PROGRAM MAIN
VAR	
	unixTime: UnixTimestamp;
	timestampNanoseconds: ULINT;

	// General variables
	mxReset									: BOOL;
	mxEmergency								: BOOL;
	EmButtons								: BOOL;
	mxAutoMode								: BOOL; (* "1" = Auto, "0" = Manual *)
	mxFirstCycle							: BOOL;
	mxErrorInit								: BOOL;
	mxInitialized							: BOOL;
	SR_AttemptedStartWithNoProductLoaded	: SR;
	
	// Sub objects
	InMoldDrying							: FB_InMoldDrying;
	ProductHandling							: FB_ProductHandling;
	Blink									: FB_Blink;

	// Variables for parameter structs and error structs
	ComSC									: ST_Com_SpeedControl;	// Communication struct for speedcontrol
	MachPar									: ST_MachPar;
	ProductPar								: ST_ProdPar;
	SysPar									: ST_SysPar;
	Errors									: ST_Errors;
	OEEpar									: ST_OEE;
	
	// Variables for/with HMI purposes
{Region "HMI variables"}
	mxHMI_Start								: BOOL;
	mxHMI_Stop								: BOOL;
	mxHMI_Pause								: BOOL;
	mxHMI_Sample							: BOOL;
	mxHMI_Reset								: BOOL;
	mxHMI_StartInit							: BOOL;
	mxHMI_StopInit							: BOOL;
	mxHMI_EnableHeating						: BOOL;

	mxHMI_StartState						: BOOL;
	mxHMI_StopState							: BOOL;
	mxHMI_PauseState						: BOOL;
	mxHMI_SampleState						: BOOL;
	mxHMI_Stopping							: BOOL;
	mxHMI_StartHydraulicsState				: BOOL;
	mxHMI_StopHydraulicsState				: BOOL;
	mxHMI_StartHydraulics					: BOOL;
	mxHMI_StopHydraulics					: BOOL;
	mxHydraulicsReady						: BOOL;
	mxProductLoaded							: BOOL;
	mxMachineInRest							: BOOL;
	
	// Speedcontrol states for hmi
	mrHMI_SpeedControlModulo				: LREAL;
	mxHMI_StartFormingPulse					: BOOL;
	mxHMI_StopFormingPulse					: BOOL;
	mxHMI_SlotANotFree						: BOOL;
	mxHMI_SlotBNotFree						: BOOL;
	mxHMI_IMDHasES							: BOOL;
	mrHMI_MaximumNrOfKickoffs				: REAL;
	mrHMI_ActNrOfKickoffs					: REAL;
	mxHMI_IMDRTO							: BOOL;
	mxHMI_IMDStopped						: BOOL;
	mxHMI_IMDRunning						: BOOL;
	mrHMI_DictatedKoSpeedControl			: LREAL;
	
	
	T_HMIReset								: TON;
	FT_AutoMode								: F_Trig;
	RT_MasterReset							: R_trig;
{End region}
	
	// Triggers for starting and stopping
	RT_Start								: R_TRIG;
	RT_Stop									: R_TRIG;
	RT_StopBySC								: R_TRIG;
	RT_StartBySC							: R_TRIG;
	RT_Pause								: R_TRIG;
	RT_StartInit							: R_TRIG;
	RT_StopInit								: R_TRIG;
	RT_StopOnLowLvl							: R_TRIG;
	RT_StartHydraulics						: R_TRIG;
	RT_StopHydraulics						: R_TRIG;	

	RT_PauseReqGantryA						: R_TRIG;
	RT_PauseReqGantryB						: R_TRIG;
	RT_PauseReqProdHandling					: R_TRIG;
	RT_PauseReqImd							: R_TRIG;
	
	// 24Volt error
	ix24VoltError1							AT %I* : BOOL;
	ix24VoltError2							AT %I* : BOOL;
	SR_24VError1							: SR;
	SR_24VError2							: SR;	
	
	// inputs and ouputs regarding safety 
{Region "Safety variables"}
	ixTwinSafe_SafetyRelay 					AT %I*:ARRAY[1..GVL.MAX_ZONES] OF BOOL; (* couple to zones in Safety programm FB outputs *)
	qxTwinSafe_Reset						AT %Q*: BOOL;
	FbError 								AT %I*: BOOL;
	ComErr 									AT %I*: BOOL;
	OutErr 									AT %I*: BOOL;
	
	(* Operator side/Front *)
	ixResetImdFront							AT %I* : BOOL;
	ixDoorReqImdFront						AT %I* : BOOL;
	qxLightEmStopImdFront					AT %Q* : BOOL;
	qxLightDoorReqImdFront					AT %Q* : BOOL;
	ixEmStopImdFront						AT %I* 	: ARRAY[0..1] OF BOOL; (* couple to the TwinSAFE inputs *)
	(* NON Operator side/Back *)
	ixResetImdBack							AT %I* : BOOL;
	ixDoorReqImdBack						AT %I* : BOOL;
	qxLightEmStopImdBack					AT %Q* : BOOL;
	qxLightDoorReqImdBack					AT %Q* : BOOL;
	ixEmStopImdBack							AT %I* 	: ARRAY[0..1] OF BOOL; (* couple to the TwinSAFE inputs *)

	(* Safety door switches *)
	ixSafetyFrontDoorLeft					AT %I* 	: ARRAY[0..1] OF BOOL; (* couple to the TwinSAFE inputs *)
	ixSafetyFrontDoorMiddle					AT %I* 	: ARRAY[0..1] OF BOOL; (* couple to the TwinSAFE inputs *)
	ixSafetyFrontDoorRight					AT %I* 	: ARRAY[0..1] OF BOOL; (* couple to the TwinSAFE inputs *)
	ixSafetyBackDoorLeft1					AT %I* 	: ARRAY[0..1] OF BOOL; (* couple to the TwinSAFE inputs *)
	ixSafetyBackDoorLeft2					AT %I* 	: ARRAY[0..1] OF BOOL; (* couple to the TwinSAFE inputs *)
	ixSafetyBackDoorMiddle3					AT %I* 	: ARRAY[0..1] OF BOOL; (* couple to the TwinSAFE inputs *)
	ixSafetyBackDoorMiddle4					AT %I* 	: ARRAY[0..1] OF BOOL; (* couple to the TwinSAFE inputs *)
	ixSafetyBackDoorRight5					AT %I* 	: ARRAY[0..1] OF BOOL; (* couple to the TwinSAFE inputs *)
	ixSafetyBackDoorRight6					AT %I* 	: ARRAY[0..1] OF BOOL; (* couple to the TwinSAFE inputs *)

	ixResetGantryA_Front					AT %I* : BOOL;
	ixDoorReqGantryA_Front					AT %I* : BOOL;
	qxLightEmStopGantryA_Front				AT %Q* : BOOL;
	qxLightDoorReqGantryA_Front				AT %Q* : BOOL;
	ixEmStopGantryA_Front					AT %I* 	: ARRAY[0..1] OF BOOL; (* couple to the TwinSAFE inputs *)

	ixResetGantryA_Back						AT %I* : BOOL;
	ixDoorReqGantryA_Back					AT %I* : BOOL;
	qxLightEmStopGantryA_Back				AT %Q* : BOOL;
	qxLightDoorReqGantryA_Back				AT %Q* : BOOL;
	ixEmStopGantryA_Back					AT %I* 	: ARRAY[0..1] OF BOOL; (* couple to the TwinSAFE inputs *)

	ixResetGantryB_Front					AT %I* : BOOL;
	ixDoorReqGantryB_Front					AT %I* : BOOL;
	qxLightEmStopGantryB_Front				AT %Q* : BOOL;
	qxLightDoorReqGantryB_Front				AT %Q* : BOOL;
	ixEmStopGantryB_Front					AT %I* 	: ARRAY[0..1] OF BOOL; (* couple to the TwinSAFE inputs *)

	ixResetGantryB_Back						AT %I* : BOOL;
	ixDoorReqGantryB_Back					AT %I* : BOOL;
	qxLightEmStopGantryB_Back				AT %Q* : BOOL;
	qxLightDoorReqGantryB_Back				AT %Q* : BOOL;
	ixEmStopGantryB_Back					AT %I* 	: ARRAY[0..1] OF BOOL; (* couple to the TwinSAFE inputs *)
	
	ixSafetyGantryA_FrontDoorLeft			AT %I* 	: ARRAY[0..1] OF BOOL; (* couple to the TwinSAFE inputs *)
	ixSafetyGantryA_FrontDoorRight			AT %I* 	: ARRAY[0..1] OF BOOL; (* couple to the TwinSAFE inputs *)
	ixSafetyGantryA_BackDoor				AT %I* 	: ARRAY[0..1] OF BOOL; (* couple to the TwinSAFE inputs *)
	ixSafetyGantryB_FrontDoorLeft			AT %I* 	: ARRAY[0..1] OF BOOL; (* couple to the TwinSAFE inputs *)
	ixSafetyGantryB_FrontDoorRight			AT %I* 	: ARRAY[0..1] OF BOOL; (* couple to the TwinSAFE inputs *)
	ixSafetyGantryB_BackDoor				AT %I* 	: ARRAY[0..1] OF BOOL; (* couple to the TwinSAFE inputs *)
{End Region}
	
	// Emergency stops
	SR_exEmergency							: ARRAY[1..GVL.MAX_ZONES] OF SR; (* Emergency of the zones *)
	SR_EmStopImdFront						: SR;
	SR_EmStopImdBack						: SR;
	SR_EmStopGantryA_Front					: SR;
	SR_EmStopGantryA_Back					: SR;
	SR_EmStopGantryB_Front					: SR;
	SR_EmStopGantryB_Back					: SR;
	
	// Emergency Doors IMD
	SR_SafetyFrontDoorLeft					: SR;
	SR_SafetyFrontDoorMiddle				: SR;
	SR_SafetyFrontDoorRight					: SR;
	SR_SafetyBackDoorLeft1					: SR;
	SR_SafetyBackDoorLeft2					: SR;
	SR_SafetyBackDoorMiddle3				: SR;
	SR_SafetyBackDoorMiddle4				: SR;
	SR_SafetyBackDoorRight5					: SR;
	SR_SafetyBackDoorRight6					: SR;
	DoorRequestImdFront						: GateRequest;
	DoorRequestImdBack						: GateRequest;
	DoorRequestGantryAFront					: GateRequest;
	DoorRequestGantryABack					: GateRequest;
	DoorRequestGantryBFront					: GateRequest;
	DoorRequestGantryBBack					: GateRequest;
	
	// Emergency Doors Gantries
	SR_SafetyGantryA_FrontDoorLeft			: SR;	
	SR_SafetyGantryA_FrontDoorRight			: SR;
	SR_SafetyGantryA_BackDoor				: SR;
	SR_SafetyGantryB_FrontDoorLeft			: SR;	
	SR_SafetyGantryB_FrontDoorRight			: SR;
	SR_SafetyGantryB_BackDoor				: SR;

	// Presistent data
	ChkMachPar								: ST_MachPar;
	CmpMachPar								: DINT;
	ChkSysPar								: ST_SysPar;
	CmpSysPar								: DINT;
	RTRIG_WritePersistent					: R_TRIG;
	FB_WritePersistentData					:  WritePersistentData;
	FB_GetCurTaskIdx						: GETCURTASKINDEX;
	T_WritePersistent						: TON;
	
	// Variables for the ethercat diagnosing.
	iwDevID									AT %I* :UINT;
	iAmsNetID								AT %I* :ARRAY [0..5] OF BYTE;
	iwSlaveCount							AT %I* :UINT;
	iwCfgSlaveCount							AT %I* :UINT;
	iwDevState								AT %I* :UINT;
	EtherCatDiag							:FB_EtherCATDiag;
	AmsNetID								: STRING;
	DeviceID								: INT;
	
	PlcCycleTime     						: REAL := 10.0;
	
	// Variables for O.E.E
	L1										AT %I* : ST_PowerMeasurement;
	L2										AT %I* : ST_PowerMeasurement;
	L3										AT %I* : ST_PowerMeasurement;	
	ActNrOfKickoffs							: REAL;	
	oldSecond								: INT;
	NTGetTime								: NT_GetTime;
	mxPulseCycle							: BOOL; 				(* Pulse 1 cycle on, 1 cycle off *)
	SysTime									: TIMESTRUCT;
	RT_1SecondTrigger						: R_TRIG;
	
	// Outputs for alarm tower.
	qxLightGreen							AT %Q* : BOOL;
	qxLightYellow							AT %Q* : BOOL;
	qxLightRed								AT %Q* : BOOL;
	qxAlarmHorn								AT %Q* : BOOL;
	
	// Variables for the UPS
	ixMainSwitchOFF							AT %I* : BOOL;	
	ixUPS_Alarm								AT %I* : BOOL;
	ixUPS_BatMode							AT %I* : BOOL;
	ixUPS_Charge							AT %I* : BOOL;
	qxPcRemoteOff							AT %Q* : BOOL;
	T_BatteryMode							: TON;
	T_MaintSwitch							: TON;
	SR_UPSAlarm								: SR;
	mxEmDoors								: BOOL;


	mxIMDUnlocked							: BOOL;
	mxProdHandlingUnlocked					: BOOL;
	mxEmptyByStopSC							: BOOL;

	RT_Sample: R_TRIG;
	mxSample: BOOL;
	RT_RestartAfterDoorOpened: R_TRIG;
	FT_Sample: F_TRIG;
	
	mxReset_ByStartInmold			: BOOL;
	mxReset_ByStartProdHandling		: BOOL;
	RT_InMoldDryingBusy				: R_TRIG;
	RT_ProdHandlingBusy				: R_TRIG;
	
	//Main Air supply
	MainAirSupply					: FB_MonoValveNoFdbck;
	MainAirPressureSwitch	AT %I* 	: BOOL;
	SR_MainAirPressureError			: SR;
	
END_VAR

unixTime();
//timestampMilliseconds := unixTime.milliseconds;
//timestampSeconds := unixTime.seconds;
timestampNanoseconds := unixTime.nanoseconds;

// 					Object Calls				//
FB_GetCurTaskIdx();
mxFirstCycle:= _TaskInfo[FB_GetCurTaskIdx.index].FirstCycle;
PlcCycleTime:= UDINT_TO_REAL(_TaskInfo[FB_GetCurTaskIdx.index].CycleTime/10000);
RemanentData();
Blink();
Objects();
HMIState();

// 					R_Trigs.					//
RT_StartHydraulics(CLK:= mxHMI_StartHydraulics);
RT_StopHydraulics(CLK:= mxHMI_StopHydraulics);
RT_Start(CLK:= mxHMI_Start);// OR (ComSC.SpeedControl_IMD.StartForming AND NOT InMoldDrying.mxInPause));
RT_Stop(CLK:= mxHMI_Stop); 
RT_StartBySC(CLK:= ComSC.SpeedControl_IMD.StartFormingA OR ComSC.SpeedControl_IMD.StartFormingB);
RT_StopBySC(CLK:= ComSC.SpeedControl_IMD.StopForming); 
RT_StopOnLowLvl(CLK:= Main.Errors.InMoldDryingErrors.ProductForming.LowLvlOnBothTanks);
RT_Pause(CLK:= mxHMI_Pause);
RT_Sample(CLK:=mxHMI_Sample);
FT_Sample(CLK:=InMoldDrying.mxSample);
RT_StartInit(CLK:= mxHMI_StartInit);
RT_StopInit(CLK:= mxHMI_StopInit);
RT_MasterReset(CLK:= NOT mxAutoMode);
mxInitialized:= InMoldDrying.mxInitialized AND ProductHandling.mxInitialized;
mxMachineInRest := NOT InMoldDrying.mxCycleBusy AND NOT ProductHandling.mxCycleBusy;


// 					Start the Hydraulics		//
IF (RT_StartHydraulics.Q OR (RT_RestartAfterDoorOpened.Q AND InMoldDrying.HydraulicsMain.mxCycleInPause AND mxAutoMode)) AND NOT mxErrorInit THEN
	InMoldDrying.M_StartHydraulics();
END_IF

// 					Stop hydraulics
IF RT_StopHydraulics.Q THEN
	InMoldDrying.M_StopHydraulics();
END_IF

RT_InMoldDryingBusy(CLK:=InMoldDrying.mxCycleBusy);
RT_ProdHandlingBusy(CLK:=ProductHandling.mxCycleBusy);
IF RT_InMoldDryingBusy.Q THEN
	mxReset_ByStartInmold := TRUE;
END_IF
IF RT_ProdHandlingBusy.Q THEN
	mxReset_ByStartProdHandling := TRUE;
END_IF
IF NOT mxEmptyByStopSC THEN
	mxReset_ByStartInmold := FALSE;
	mxReset_ByStartProdHandling := FALSE;	
END_IF

// 					Start machine				//
IF (RT_Start.Q OR (mxEmptyByStopSC AND NOT ComSC.SpeedControl_IMD.StopForming)) AND mxAutoMode AND mxInitialized AND NOT mxErrorInit AND mxProductLoaded AND mxHydraulicsReady AND NOT mxIMDUnlocked AND NOT mxProdHandlingUnlocked THEN  
	InMoldDrying.M_StartCycle(); 
	ProductHandling.M_StartCycle();
	mxHMI_Stopping :=FALSE;
	IF mxReset_ByStartInmold AND mxReset_ByStartProdHandling THEN
		mxEmptyByStopSC := FALSE;
	END_IF
END_IF

//					IMD Pause (stopinpos)		//
IF RT_PauseReqImd.Q THEN
	InMoldDrying.M_StopCycle();	
	mxEmptyByStopSC := FALSE;
END_IF

//					Producthandling Pause (stopinpos)		//
IF RT_PauseReqProdHandling.Q THEN
	ProductHandling.M_StopCycle();	
	mxEmptyByStopSC := FALSE;
END_IF

//					Normal stop					//
IF ((RT_StopOnLowLvl.Q OR RT_Stop.Q OR RT_StopBySC.Q) AND mxAutoMode) THEN  
	InMoldDrying.M_StopCycleEmpty();  
	Producthandling.M_StopCycleEmpty(); 
	mxHMI_Stopping := TRUE;		
	mxEmptyByStopSC := FALSE;
	IF 	RT_StopBySC.Q AND (ProductHandling.mxCycleBusy OR InMoldDrying.mxCycleBusy) THEN
		mxEmptyByStopSC := TRUE;
	END_IF			
END_IF

//					Init machine				//
IF RT_StartInit.Q AND mxAutoMode AND mxProductLoaded AND NOT mxErrorInit AND mxHydraulicsReady THEN 
	InMoldDrying.M_StartInit(); 
	mxEmptyByStopSC := FALSE;
	Producthandling.M_StartInit(); 
END_IF
IF RT_StopInit.Q OR mxErrorInit THEN
	InMoldDrying.M_StopInit();
	ProductHandling.M_StopInit();
	mxEmptyByStopSC := FALSE;
END_IF

//					Stop direct error			//
IF mxErrorInit OR InMoldDrying.mxErrorInit OR ProductHandling.Errors.Gantry_A.Collision OR ProductHandling.Errors.Gantry_B.Collision THEN
	InMoldDrying.M_StopDirect();
	mxEmptyByStopSC := FALSE;
END_IF

IF mxErrorInit OR ProductHandling.mxErrorInit THEN
	ProductHandling.M_StopDirect();
	mxEmptyByStopSC := FALSE;
END_IF



//					Signal light				//
qxLightEmStopImdFront:= qxLightEmStopImdBack:= qxLightEmStopGantryA_Front:= qxLightEmStopGantryA_Back:= qxLightEmStopGantryB_Front:= qxLightEmStopGantryB_Back := 
	Errors.exEmergency[1] OR Errors.exEmergency[2] OR Errors.exEmergency[3] OR Errors.exEmergency[4] OR Errors.exEmergency[5] OR Errors.exEmergency[6] OR Errors.exEmergency[7];
qxLightRed:= HMI.mxError;
qxLightGreen:= mxHMI_StartState := (InMoldDrying.mxCycleBusy OR ProductHandling.mxCycleBusy) AND NOT mxHMI_PauseState;
qxLightYellow:= FALSE;

//					Reseting					//
T_HMIReset(IN:= mxHMI_Reset,PT:=T#1S);
IF T_hmiReset.Q THEN mxHMI_Reset:=FALSE; END_IF

mxReset:= qxTwinSafe_Reset:= mxHMI_Reset OR ixResetImdFront OR ixResetImdBack OR ixResetGantryA_Front OR ixResetGantryA_Back OR ixResetGantryB_Front OR ixResetGantryB_Back;

//					Master reset				//
IF RT_MasterReset.Q THEN
	InMoldDrying.mxResetCycleState := TRUE;
	InMoldDrying.mxResetInitState := TRUE;
	ProductHandling.mxResetCycleState:= TRUE;
	ProductHandling.mxResetInitState:= TRUE;
	mxEmptyByStopSC := FALSE;
END_IF

// 					Sample button				//
IF RT_Sample.Q THEN
	mxSample:= InMoldDrying.mxSample := TRUE;
END_IF; 

IF FT_Sample.Q THEN
	mxSample:=FALSE;
END_IF


// Get AMS net id and device id for ethercat topology
AmsNetID:= F_CreateAmsNetId(iAmsNetID);
DeviceID:= UINT_TO_INT(iwDevID);

// 					Force HMI bits to zero		//
mxHMI_Start := FALSE;
mxHMI_Stop := FALSE;
mxHMI_Pause := FALSE;
mxHMI_Sample:=FALSE;
mxHMI_StartHydraulics := FALSE;
mxHMI_StopHydraulics:=FALSE;

// Shut of PC when on battery mode or when power was switched off:
T_BatteryMode(IN:=ixUPS_BatMode, PT:=T#30S);
T_MaintSwitch(IN:=ixMainSwitchOFF, PT:=T#5S);

// Uncomment when timers are tested.
qxPcRemoteOff := T_BatteryMode.Q OR T_MaintSwitch.Q;

//Main Air Supply
MainAirSupply.M_On();

ACTION Com_SC:
// Current speed (dictated by Speedcontrol)
IF InMoldDrying.ProductForming.CurrentSpeedSingleKO > 0 THEN
	ComSC.IMD_SpeedControl.ActualSpeed := (60000 / InMoldDrying.ProductForming.CurrentSpeedSingleKO);
END_IF

// Current maximum speed (Calculated on bases of own forming).
ComSC.IMD_SpeedControl.MaximumSpeed := InMoldDrying.CalculateMaxKO.MaxKO;


ComSC.IMD_SpeedControl.RTO := mxAutoMode AND mxInitialized AND NOT mxErrorInit AND mxProductLoaded AND mxHydraulicsReady;
ComSC.IMD_SpeedControl.ES := mxEmergency;
ComSC.IMD_SpeedControl.Stopped := NOT InMoldDrying.mxCycleBusy; // AND NOT ProductHandling.mxCycleBusy;
ComSC.IMD_SpeedControl.HMI_Reset := mxHMI_Reset;
END_ACTION

ACTION Error:
(*Emergency Stop Active Zone x,  Index=Zone , 1=Takeout/Gantr A, 2=Imd Left, 3=Imd Middle, 4=Imd Right, 5=Takeout/Gantry B*, 6=Gantry B *)
SR_exEmergency[1](SET1:= NOT ixTwinSafe_SafetyRelay[1], RESET:=ixTwinSafe_SafetyRelay[1] , Q1=>Errors.exEmergency[1] );
SR_exEmergency[2](SET1:= NOT ixTwinSafe_SafetyRelay[2], RESET:=ixTwinSafe_SafetyRelay[2] , Q1=>Errors.exEmergency[2] );
SR_exEmergency[3](SET1:= NOT ixTwinSafe_SafetyRelay[3], RESET:=ixTwinSafe_SafetyRelay[3] , Q1=>Errors.exEmergency[3] );
SR_exEmergency[4](SET1:= NOT ixTwinSafe_SafetyRelay[4], RESET:=ixTwinSafe_SafetyRelay[4] , Q1=>Errors.exEmergency[4] );
SR_exEmergency[5](SET1:= NOT ixTwinSafe_SafetyRelay[5] , RESET:=ixTwinSafe_SafetyRelay[5], Q1=>Errors.exEmergency[5] );
SR_exEmergency[6](SET1:= NOT ixTwinSafe_SafetyRelay[6] , RESET:=ixTwinSafe_SafetyRelay[6], Q1=>Errors.exEmergency[6] );
SR_exEmergency[7](SET1:= NOT ixTwinSafe_SafetyRelay[7] , RESET:=ixTwinSafe_SafetyRelay[7], Q1=>Errors.exEmergency[7] );

(*InMold Drying *)
SR_EmStopImdFront(SET1:= NOT ixEmStopImdFront[0] OR NOT ixEmStopImdFront[1] , RESET:= mxReset, Q1=> Errors.exEmStopImdFront);
SR_EmStopImdBack(SET1:= NOT ixEmStopImdBack[0] OR NOT ixEmStopImdBack[1] , RESET:= mxReset, Q1=> Errors.exEmStopImdBack);

SR_SafetyFrontDoorLeft(SET1:= NOT ixSafetyFrontDoorLeft[0] OR NOT ixSafetyFrontDoorLeft[1] , RESET:= mxReset, Q1=> Errors.exImdFrontDoorLeft);
SR_SafetyFrontDoorMiddle(SET1:= NOT ixSafetyFrontDoorMiddle[0] OR NOT ixSafetyFrontDoorMiddle[1] , RESET:= mxReset, Q1=> Errors.exImdFrontDoorMiddle);
SR_SafetyFrontDoorRight(SET1:= NOT ixSafetyFrontDoorRight[0] OR NOT ixSafetyFrontDoorRight[1] , RESET:= mxReset, Q1=> Errors.exImdFrontDoorRight);
SR_SafetyBackDoorLeft1(SET1:= NOT ixSafetyBackDoorLeft1[0] OR NOT ixSafetyBackDoorLeft1[1] , RESET:= mxReset, Q1=> Errors.exImdBackDoorLeft1);
SR_SafetyBackDoorLeft2(SET1:= NOT ixSafetyBackDoorLeft2[0] OR NOT ixSafetyBackDoorLeft2[1] , RESET:= mxReset, Q1=> Errors.exImdBackDoorLeft2);
SR_SafetyBackDoorMiddle3(SET1:= NOT ixSafetyBackDoorMiddle3[0] OR NOT ixSafetyBackDoorMiddle3[1] , RESET:= mxReset, Q1=> Errors.exImdBackDoorMiddle3);
SR_SafetyBackDoorMiddle4(SET1:= NOT ixSafetyBackDoorMiddle4[0] OR NOT ixSafetyBackDoorMiddle4[1] , RESET:= mxReset, Q1=> Errors.exImdBackDoorMiddle4);
SR_SafetyBackDoorRight5(SET1:= NOT ixSafetyBackDoorRight5[0] OR NOT ixSafetyBackDoorRight5[1] , RESET:= mxReset, Q1=> Errors.exImdBackDoorRight5);
SR_SafetyBackDoorRight6(SET1:= NOT ixSafetyBackDoorRight6[0] OR NOT ixSafetyBackDoorRight6[1] , RESET:= mxReset, Q1=> Errors.exImdBackDoorRight6);

(* Gantry *)
SR_EmStopGantryA_Front(SET1:= NOT ixEmStopGantryA_Front[0] OR NOT ixEmStopGantryA_Front[1] ,RESET:= mxReset, Q1=> Errors.exEmStopGantryA_Front);
SR_EmStopGantryA_Back(SET1:= NOT ixEmStopGantryA_Back[0] OR NOT ixEmStopGantryA_Back[1] ,RESET:= mxReset, Q1=> Errors.exEmStopGantryA_Back);
SR_EmStopGantryB_Front(SET1:= NOT ixEmStopGantryB_Front[0] OR NOT ixEmStopGantryB_Front[1] ,RESET:= mxReset, Q1=> Errors.exEmStopGantryB_Front);
SR_EmStopGantryB_Back(SET1:= NOT ixEmStopGantryB_Back[0] OR NOT ixEmStopGantryB_Back[1] ,RESET:= mxReset, Q1=> Errors.exEmStopGantryB_Back);

SR_SafetyGantryA_FrontDoorLeft(SET1:= NOT ixSafetyGantryA_FrontDoorLeft[0] OR NOT ixSafetyGantryA_FrontDoorLeft[1] , RESET:= mxReset, Q1=> Errors.exGantryA_FrontDoorLeft);
SR_SafetyGantryA_FrontDoorRight(SET1:= NOT ixSafetyGantryA_FrontDoorRight[0] OR NOT ixSafetyGantryA_FrontDoorright[1] , RESET:= mxReset, Q1=> Errors.exGantryA_FrontDoorRight);
SR_SafetyGantryA_BackDoor(SET1:= NOT ixSafetyGantryA_BackDoor[0] OR NOT ixSafetyGantryA_BackDoor[1] , RESET:= mxReset, Q1=> Errors.exGantryA_BackDoor);
SR_SafetyGantryB_FrontDoorLeft(SET1:= NOT ixSafetyGantryB_FrontDoorLeft[0] OR NOT ixSafetyGantryB_FrontDoorLeft[1] , RESET:= mxReset, Q1=> Errors.exGantryB_FrontDoorLeft);
SR_SafetyGantryB_FrontDoorRight(SET1:= NOT ixSafetyGantryB_FrontDoorRight[0] OR NOT ixSafetyGantryB_FrontDoorright[1] , RESET:= mxReset, Q1=> Errors.exGantryB_FrontDoorRight);
SR_SafetyGantryB_BackDoor(SET1:= NOT ixSafetyGantryB_BackDoor[0] OR NOT ixSafetyGantryB_BackDoor[1] , RESET:= mxReset, Q1=> Errors.exGantryB_BackDoor);

(* Main Air Supply *)
SR_MainAirPressureError(SET1 := NOT MainAirPressureSwitch, RESET:= mxReset, Q1=> Errors.MainAirSupplyError);

(*24V error*)
SR_24VError1(Set1:=NOT ix24VoltError1, Reset:=mxReset, Q1=>Errors.ex24VoltError1); 
SR_24VError2(Set1:=NOT ix24VoltError2, Reset:=mxReset, Q1=>Errors.ex24VoltError2); 
SR_UPSAlarm(Set1:=NOT ixUPS_Alarm, Reset:=mxReset, Q1=>Errors.exUpsAlarm);

SR_AttemptedStartWithNoProductLoaded(Set1:=NOT mxProductLoaded AND (RT_Start.Q OR RT_StartInit.Q), Reset:=mxReset, Q1=>Errors.exAtteptedStartWithNoProduct);

EtherCatDiag(
	SlaveCount:=	iwSlaveCount,
	CfgSlaveCount:=	iwCfgSlaveCount,
	DevState:=		iwDevState);

Errors.exEmergency[8]	:=EmButtons := Errors.exEmStopGantryA_Back OR Errors.exEmStopGantryA_Front OR Errors.exEmStopGantryB_Back OR Errors.exEmStopGantryB_Front OR Errors.exEmStopImdBack OR Errors.exEmStopImdFront;

mxEmDoors	:= Errors.exEmergency[1] OR Errors.exEmergency[2] OR Errors.exEmergency[3] OR 
Errors.exEmergency[4] OR Errors.exEmergency[5] OR Errors.exEmergency[6] OR Errors.exEmergency[7]; 	

mxEmergency := mxEmDoors OR EmButtons;

mxErrorInit:= InMoldDrying.mxErrorInit OR ProductHandling.mxErrorInit OR EmButtons OR Errors.MainAirSupplyError OR
				(NOT InMoldDrying.mxInPause AND NOT ProductHandling.mxInPause AND mxEmDoors); // If door is opened without door req, stopdirect (mxErrorInit).
END_ACTION

ACTION HMIState:
//// ***			Starting stopping pause Sample			***	////
mxHMI_StartHydraulicsState := mxHydraulicsReady;
mxHMI_StopHydraulicsState := NOT mxHydraulicsReady;
mxHMI_StartState:= InMoldDrying.mxCycleBusy AND ProductHandling.mxCycleBusy;
mxHMI_PauseState:= InMoldDrying.mxInPause AND ProductHandling.mxInPause;
mxHMI_StopState:= (NOT InMoldDrying.mxCycleBusy AND NOT ProductHandling.mxCycleBusy) OR mxHMI_Stopping;
mxHMI_IMDRunning := NOT mxHMI_PauseState AND (InMoldDrying.mxCycleBusy OR ProductHandling.mxCycleBusy);
mxHMI_SampleState := mxSample;


//// *** 					Speedcontrol					*** ////

// Status for HMI: Speedcontrol commands for IMD
mrHMI_SpeedControlModulo := ComSC.SpeedControl_IMD.Modulo;
mxHMI_StartFormingPulse := ComSC.SpeedControl_IMD.StartFormingA OR ComSC.SpeedControl_IMD.StartFormingB;
mxHMI_StopFormingPulse := ComSC.SpeedControl_IMD.StopForming;
mxHMI_SlotANotFree := ComSc.SpeedControl_IMD.ErrSlotANotFree;
mxHMI_SlotBNotFree := ComSc.SpeedControl_IMD.ErrSlotBNotFree;

// Status for HMI: IMD commands for Speedcontrol
mxHMI_ImdHasES := ComSC.IMD_SpeedControl.ES;
mrHMI_ActNrOfKickoffs := ComSC.IMD_SpeedControl.ActualSpeed;
mrHMI_MaximumNrOfKickoffs := ComSc.IMD_SpeedControl.MaximumSpeed;
mxHMI_IMDRTO := ComSc.IMD_SpeedControl.RTO;
mxHMI_IMDStopped := ComSC.IMD_SpeedControl.Stopped;
mrHMI_DictatedKoSpeedControl := ComSC.SpeedControl_IMD.SpeedInKo;
END_ACTION

ACTION Objects:
HMI();
Error();
SafetyDoors();
Com_SC();
OEE();

InMoldDrying(
	mxReset:= mxReset, 
	mxEmergency:= Errors.exEmergency,//Errors.exEmergency[1] OR Errors.exEmergency[2] OR Errors.exEmergency[3] OR Errors.exEmergency[4] OR Errors.exEmergency[5] OR Errors.exEmStopImdFront OR Errors.exEmStopImdBack,
	mxAutoMode:= mxAutoMode,
	mxStartFormingA:= ComSC.SpeedControl_IMD.StartFormingA,
	mxStartFormingB:= ComSC.SpeedControl_IMD.StartFormingB,
	mxFirstCycle:= mxFirstCycle,
	mxProductPickedUpGantry_A:= ProductHandling.mxProductPickedUpGantry_A,
	mxProductPickedUpGantry_B:= ProductHandling.mxProductPickedUpGantry_B,
	mxEnableHeating:= mxHMI_EnableHeating,
	mxHydraulicsReady=>mxHydraulicsReady,
	mxGantrysNotBusy:= ProductHandling.mxGantrysNotBusy,
	PlcCycleTime:=PlcCycleTime,
	MachParameters:= MachPar.InMoldDrying, 
	ProdParameters:= ProductPar.InMoldDrying, 
	SysParameters:= SysPar.InMoldDrying,
	mxFormingA_Ready => ComSC.IMD_SpeedControl.FormingReadyA,
	mxFormingB_Ready => ComSC.IMD_SpeedControl.FormingReadyB,
	Errors=> Errors.InMoldDryingErrors);

ProductHandling(
	mxReset:= mxReset, 
	mxEmergency:= Errors.exEmergency,//Errors.exEmergency[1] OR Errors.exEmergency[5] OR Errors.exEmergency[6] OR Errors.exEmergency[7] OR Errors.exEmStopImdFront OR Errors.exEmStopImdBack,
	mxAutoMode:= mxAutoMode,
	mxFirstCycle:=mxFirstCycle,
	mxSideA_Enabled:= InMoldDrying.mxSideAEnabled, //MachPar.InMoldDrying.EnableEamcSideA,
	mxSideB_Enabled:= InMoldDrying.mxSideBEnabled, //MachPar.InMoldDrying.EnableEamcSideB,
	mxEamcIsEmpty:= InMoldDrying.mxIsEmpty,
	mxStopBeforeSCstarted := InMoldDrying.mxStopBeforeSCstarted,
	mxProductReadyAtTakeout_A:= InMoldDrying.mxProductReadyAtTakeout_A,
	mxProductReadyAtTakeout_B:= InMoldDrying.mxProductReadyAtTakeout_B,
	mxStopCycleGantryA:=RT_PauseReqGantryA.Q,
	mxStopCycleGantryB:=RT_PauseReqGantryB.Q,
	GantryA_BlowOffPulse:= ComSC.SpeedControl_IMD.BlowOffPulseA,
	GantryB_BlowOffPulse:= ComSC.SpeedControl_IMD.BlowOffPulseB,
	GantryA_BlowOffSucceded	=> ComSC.IMD_SpeedControl.BlowOffProcessedA,
	GantryB_BlowOffSucceded	=> ComSC.IMD_SpeedControl.BlowOffProcessedB,
	GantryA_InPositionAtBelt=> ComSC.IMD_SpeedControl.GantryA_Ready,
	GantryB_InPositionAtBelt=> ComSC.IMD_SpeedControl.GantryB_Ready,
	NrOfSheets := ComSC.SpeedControl_IMD.ProdParameters.NrOfSheets,
	NrOfCavities := COmSC.SpeedControl_IMD.ProdParameters.NrOfCavities,
	MachParameters:= MachPar.ProductHandling, 
	ProdParameters:= ProductPar.ProductHandling,
	SysParameters:= SysPar.ProductHandling,
	Errors=> Errors.ProductHandlingErrors);

MainAirSupply(
	mxReset:= mxReset, 
	mxEmergency:= , 
	mxAutoMode:= TRUE, 
	RHSR_Blocked:= , 
	SlowValveIsInverted:= , 
	mxDisableManualAutoTrigger:= , 
	mxIsOn=> );
END_ACTION

ACTION OEE:
(* Read actual Systemtime *)
mxPulseCycle := NOT mxPulseCycle;
NTGetTime(START:=mxPulseCycle AND NOT NTGetTime.BUSY , TMOUT:=t#100ms,  TIMESTR=>SysTime );

RT_1SecondTrigger(CLK:=WORD_TO_INT(SysTime.wSecond) <> oldSecond);
IF RT_1SecondTrigger.Q THEN
	oldSecond:=WORD_TO_INT(SysTime.wSecond);
END_IF

// Calculate the voltage to normal format (000.00V)
OEEpar.L1_Voltage := DINT_TO_REAL(L1.iwVoltage) / 10000.0;
OEEpar.L2_Voltage := DINT_TO_REAL(L2.iwVoltage) / 10000.0;
OEEpar.L3_Voltage := DINT_TO_REAL(L3.iwVoltage) / 10000.0;

// Calculate the current to normal format (00.00A)
OEEpar.L1_Current := DINT_TO_REAL(L1.iwCurrent) / 1000.0;
OEEpar.L2_Current := DINT_TO_REAL(L2.iwCurrent) / 1000.0;
OEEpar.L3_Current := DINT_TO_REAL(L3.iwCurrent) / 1000.0;

// Calculate the Powerconsumtion 
OEEpar.L1_Watt := OEEpar.L1_Voltage * OEEpar.L1_Current;
OEEpar.L2_Watt := OEEpar.L2_Voltage * OEEpar.L2_Current;
OEEpar.L3_Watt := OEEpar.L3_Voltage * OEEpar.L3_Current;

// Kickoff's A side
IF InMoldDrying.BottommoldA.NrOfKickOffs <> 0 THEN
	OEEpar.KickOffsAside := (60000 / InMoldDrying.BottommoldA.NrOfKickOffs);
ELSE
	OEEpar.KickOffsAside := 0;
END_IF

// Kickoff's B side
IF InMoldDrying.BottommoldB.NrOfKickOffs <> 0 THEN
	OEEpar.KickOffsBside := (60000 / InMoldDrying.BottommoldB.NrOfKickOffs);
ELSE
	OEEpar.KickOffsBside := 0;
END_IF

// Total Kickoff's
OEEpar.KickOffsBothSides := ComSC.IMD_SpeedControl.ActualSpeed;

// IMD Error time:
IF RT_1SecondTrigger.Q AND (InMoldDrying.mxErrorInit OR InMoldDrying.mxErrorStopinPos) THEN
	OEEpar.ImdErrorTime := OEEpar.ImdErrorTime +1;
END_IF

// ProductHandling Error Time:
IF RT_1SecondTrigger.Q AND (ProductHandling.mxErrorInit OR ProductHandling.mxErrorStopinPos) THEN
	OEEpar.ProductHandingErrorTime := OEEpar.ProductHandingErrorTime +1;
END_IF

// Total run time (time that the machine was in automatic production mode)
IF RT_1SecondTrigger.Q AND (mxAutomode AND mxHMI_IMDRunning) THEN
	OEEpar.TotalRunTime := OEEpar.TotalRunTime +1;
END_IF

// Total wait time (time that the machine was ready, with no error, but wasn't running)
IF RT_1SecondTrigger.Q AND (mxAutomode AND NOT mxHMI_IMDRunning AND mxInitialized) THEN
	OEEpar.TotalWaitTime := OEEpar.TotalWaitTime +1;
END_IF

// Down time (time that the machine was unable to operate cause of an error).
// Total wait time (time that the machine was ready, with no error, but wasn't running)
IF RT_1SecondTrigger.Q AND (mxAutomode AND NOT mxHMI_IMDRunning AND (InMoldDrying.mxErrorInit OR InMoldDrying.mxErrorStopinPos OR 
ProductHandling.mxErrorInit OR ProductHandling.mxErrorStopinPos)) THEN
	OEEpar.TotalDownTime := OEEpar.TotalDownTime +1;
END_IF

// Products for A.
OEEpar.ProducedSheetsASide := Main.MachPar.ProductHandling.GantryA.SheetsProduced;			// Number of sheets that the A side has produced
OEEpar.ProducedProductsAside := Main.MachPar.ProductHandling.GantryA.ProductsProduced;			// Number of Products that the A side has produced

// Products for A.
OEEpar.ProducedSheetsBSide := Main.MachPar.ProductHandling.GantryB.SheetsProduced;			// Number of sheets that the B side has produced
OEEpar.ProducedProductsBside := Main.MachPar.ProductHandling.GantryB.ProductsProduced;			// Number of Products that the B side has produced

// Total produced sheets and products.
OEEpar.TotalProducedSheets := Main.MachPar.ProductHandling.GantryA.SheetsProduced + Main.MachPar.ProductHandling.GantryB.SheetsProduced;	
OEEpar.TotalProducedProducts := Main.MachPar.ProductHandling.GantryA.ProductsProduced + Main.MachPar.ProductHandling.GantryB.ProductsProduced;
END_ACTION

ACTION RemanentData:
IF mxFirstCycle THEN
	MachPar:= PersMachPar;
	SysPar:= PersSysPar;
END_IF

CmpMachPar:= MEMCMP(ADR(MachPar), ADR(ChkMachPar),SIZEOF(ChkMachPar));
CmpSysPar:= MEMCMP(ADR(SysPar), ADR(ChkSysPar),SIZEOF(ChkSysPar));

(* Backup every x min. the persistent parameters *)
T_WritePersistent(IN:= NOT T_WritePersistent.Q , PT:=T#5M);

RTrig_WritePersistent(CLK:= (CmpMachPar <> 0) OR (CmpSysPar <> 0));

IF RTRIG_WritePersistent.Q THEN
	PersMachPar:= MachPar;
	PersSysPar:= SysPar;
	FB_WritePersistentData(NETID:='', PORT:=851, START:=TRUE, TMOUT:=T#1S );	
ELSE
	FB_WritePersistentData(NETID:='', PORT:=851, START:=FALSE, TMOUT:=T#1S );
END_IF

ChkMachPar:= MachPar;
ChkSysPar:= SysPar;
END_ACTION

ACTION SafetyDoors:
{Region "In mold dryer doors"} 
// In mold dryer 
DoorRequestImdFront(
	GateClosed:= NOT Errors.exImdFrontDoorLeft AND NOT Errors.exImdFrontDoorMiddle AND NOT Errors.exImdFrontDoorRight, 
	SafeState:= InMoldDrying.mxInPause AND ProductHandling.mxInPause, 
	Request_Open:= ixDoorReqImdFront, 
	Reset:=mxReset, 
	TimeOutSafeState:= T#10S, 
	Lock=> , 
	GateRequest_Light=> qxLightDoorReqImdFront, 
	ResetButton_Light=> );

DoorRequestImdBack(
	GateClosed:= NOT Errors.exImdBackDoorLeft1 AND NOT Errors.exImdBackDoorLeft2 AND NOT Errors.exImdBackDoorMiddle3 AND NOT Errors.exImdBackDoorMiddle4 
	AND NOT Errors.exImdBackDoorRight5 AND NOT errors.exImdBackDoorRight6, 
	SafeState:= InMoldDrying.mxInPause AND ProductHandling.mxInPause, 
	Request_Open:= ixDoorReqImdBack, 
	Reset:=mxReset, 
	TimeOutSafeState:= T#10S, 
	Lock=> , 
	GateRequest_Light=> qxLightDoorReqImdBack, 
	ResetButton_Light=> );
{End Region}
	
{Region "Gantries"}
// Gantry A Front
DoorRequestGantryAFront(
	GateClosed:= NOT Errors.exGantryA_FrontDoorLeft AND NOT Errors.exGantryA_FrontDoorRight, 
	SafeState:= InMoldDrying.mxInPause AND ProductHandling.mxInPause,  
	Request_Open:= ixDoorReqGantryA_Front, 
	Reset:=mxReset, 
	TimeOutSafeState:= T#10S, 
	Lock=> , 
	GateRequest_Light=> qxLightDoorReqGantryA_Front, 
	ResetButton_Light=> );

DoorRequestGantryABack(
	GateClosed:= NOT Errors.exGantryA_BackDoor, 
	SafeState:= InMoldDrying.mxInPause AND ProductHandling.mxInPause,  
	Request_Open:= ixDoorReqGantryA_Back, 
	Reset:=mxReset, 
	TimeOutSafeState:= T#10S, 
	Lock=> , 
	GateRequest_Light=> qxLightDoorReqGantryA_Back, 
	ResetButton_Light=> );

DoorRequestGantryBFront(
	GateClosed:= NOT Errors.exGantryB_FrontDoorLeft AND NOT Errors.exGantryB_FrontDoorRight, 
	SafeState:= InMoldDrying.mxInPause AND ProductHandling.mxInPause, 
	Request_Open:= ixDoorReqGantryB_Front, 
	Reset:=mxReset, 
	TimeOutSafeState:= T#10S, 
	Lock=> , 
	GateRequest_Light=> qxLightDoorReqGantryB_Front, 
	ResetButton_Light=> );
	
DoorRequestGantryBBack(
	GateClosed:= NOT Errors.exGantryB_BackDoor, 
	SafeState:= InMoldDrying.mxInPause AND ProductHandling.mxInPause, 
	Request_Open:= ixDoorReqGantryB_Back, 
	Reset:=mxReset, 
	TimeOutSafeState:= T#10S, 
	Lock=> , 
	GateRequest_Light=> qxLightDoorReqGantryB_Back, 
	ResetButton_Light=> );
{End Region}

// Collect al lockstates.
mxIMDUnlocked := NOT DoorRequestImdFront.Lock OR NOT DoorRequestImdBack.Lock;
mxProdHandlingUnlocked := NOT DoorRequestGantryABack.Lock OR NOT DoorRequestGantryAFront.Lock OR NOT DoorRequestGantryBBack.Lock OR NOT DoorRequestGantryBFront.Lock;
RT_RestartAfterDoorOpened(CLK:=NOT mxIMDUnlocked AND NOT mxProdHandlingUnlocked AND mxReset);


// Handle the requests
RT_PauseReqImd(ClK:=(ixDoorReqImdFront OR ixDoorReqImdBack OR ixDoorReqGantryA_Front OR ixDoorReqGantryB_Front OR InMoldDrying.mxErrorStopinPos) AND mxAutoMode);
//RT_PauseReqGantryA(CLK:=ixDoorReqImdFront OR ixDoorReqImdBack OR ixDoorReqGantryA_Front OR ixDoorReqGantryA_Back);
//RT_PauseReqGantryB(CLK:=ixDoorReqImdFront OR ixDoorReqImdBack OR ixDoorReqGantryB_Front OR ixDoorReqGantryB_Back);
RT_PauseReqProdHandling(CLK:=(ixDoorReqImdFront OR ixDoorReqImdBack OR ixDoorReqGantryB_Front OR ixDoorReqGantryB_Back OR InMoldDrying.mxErrorStopinPos)AND mxAutoMode);
END_ACTION

END_PROGRAM

(* stored: Version 1.1.0.1, ProductVersion 3.1.4022.16
   POU MAIN: Id {147bab3f-acfd-4acf-8d8e-a76750ccc81a}, SpecialFunc None
   Action Com_SC: Id {d783749b-6813-4311-9fc2-4a90fec2a0cc}
   Action Error: Id {32a11183-149e-4a28-9cb7-3681850f3bf8}
   Action HMIState: Id {3b6d2f35-c3dd-4e70-be6d-7a184a0192e1}
   Action Objects: Id {2a794986-d238-4cdf-83df-adb4601c4b15}
   Action OEE: Id {b9d6c661-be12-4631-a38e-4ad57534fc61}
   Action RemanentData: Id {c93fd129-2948-45c7-836c-2640a4ab3350}
   Action SafetyDoors: Id {44b09eb6-68f0-4032-a64c-9a91aaa03aa3} *)
